ABB RobotStudio station: zaliczenie_zadanie2_20200112-154802.rsstn

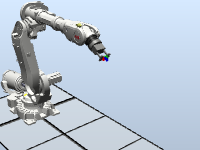
Station zaliczenie_zadanie2 (saved by RobotStudio 6.8.8307.1040)
Controller IRB_6640_185kg_2.80m
  mechanical unit ROB_1: IRB6640_185_280__04, 6 joints, base frame (0, 0, 0) mm
Layout (positions relative to the parent item):
  - IRB6640_185_280__04 [mechanism, from Robots\IRB6640_185_280_G_04.rslib] at (0, 0, 0) mm; joint values [0, 0, 0, 0, 0.5236, 0] (rad or m)
  - rence_bonczura [mechanism] at (1885.71, 0, 1955) mm, rotated rx 180 ry 60 rz 180 deg; joint values [0, 0] (rad or m)
      TCP rence_bonczura_1 at (0, 0, 260) mm
      links: base, left, right
Attachment: rence_bonczura is attached to IRB6640_185_280__04 / Link6
Targets, tools, work objects and paths stored in the station, written as RAPID:
! task T_ROB1
MODULE CalibData
  PERS tooldata rence_bonczura_1:=[TRUE,[[0,0,260],[1,0,0,0]],[1,[1,1,1],[1,0,0,0],0,0,0]];
ENDMODULE

